// TIA Portal V17 export
// export: Created 2025-03-07T09:23:50.1385037Z, ExportSetting WithDefaults, DisplayName Totally Integrated Automation Portal, DisplayVersion V17 Update 8, DisplayName TIA Portal Openness, DisplayVersion V17 Update 8, DisplayName TIA Portal Version Control Interface, DisplayVersion V17, DisplayName SINAMICS Startdrive Advanced, DisplayVersion V17 SP2, DisplayName SINAMICS Startdrive G110M, G120, G120C, G120D, G120P, G115D, DisplayVersion V17 SP2, DisplayName SINAMICS Startdrive G130, G150, S120, S150, SINAMICS MV, S210, DisplayVersion V17 SP2, DisplayName STEP 7 Professional, DisplayVersion V17 Update 8, DisplayName SINUMERIK ONE STEP 7 Toolbox, DisplayVersion V17 Update 12, DisplayName SINUMERIK 840D sl STEP 7 Toolbox, DisplayVersion V17 Update 12, DisplayName STEP 7 Safety, DisplayVersion V17 Update 6, DisplayName WinCC Advanced, DisplayVersion V17 Update 8
FUNCTION "FC7341_MACHINE_TO_POWDER_INTERLOCK" : Void   // FC7341, LAD
{ S7_Optimized_Access := 'TRUE' }
VERSION : 0.1
// stored: AutoNumber false, IsIECCheckEnabled false, SetENOAutomatically false, UDAEnableTagReadback false
   VAR_TEMP
      "COUNT_FOR _ERROR" : Int;
      EKS_IDENT : Array[0..7] of Char;   // EKS OPERATOR ID
   END_VAR
   VAR CONSTANT
      FC_NUMBER : DInt := 7341;
   END_VAR
BEGIN

REGION Network 1: //////////_GENERAL_//////////
END_REGION

REGION Network 2: LIFE BIT
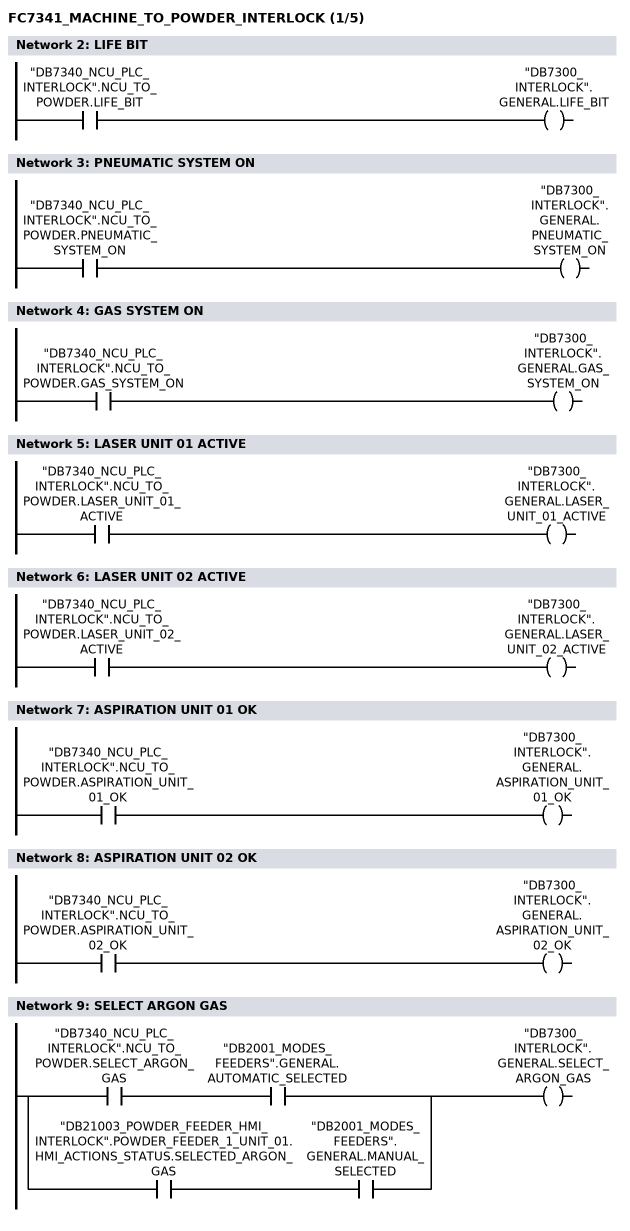
   RUNG wire#powerrail
      Contact( "DB7340_NCU_PLC_INTERLOCK".NCU_TO_POWDER.LIFE_BIT )
      Coil( "DB7300_INTERLOCK".GENERAL.LIFE_BIT )
   END_RUNG
   // the same network as SCL:
   "DB7300_INTERLOCK".GENERAL.LIFE_BIT := "DB7340_NCU_PLC_INTERLOCK".NCU_TO_POWDER.LIFE_BIT;
END_REGION

REGION Network 3: PNEUMATIC SYSTEM ON
   RUNG wire#powerrail
      Contact( "DB7340_NCU_PLC_INTERLOCK".NCU_TO_POWDER.PNEUMATIC_SYSTEM_ON )
      Coil( "DB7300_INTERLOCK".GENERAL.PNEUMATIC_SYSTEM_ON )
   END_RUNG
   // the same network as SCL:
   "DB7300_INTERLOCK".GENERAL.PNEUMATIC_SYSTEM_ON := "DB7340_NCU_PLC_INTERLOCK".NCU_TO_POWDER.PNEUMATIC_SYSTEM_ON;
END_REGION

REGION Network 4: GAS SYSTEM ON
   RUNG wire#powerrail
      Contact( "DB7340_NCU_PLC_INTERLOCK".NCU_TO_POWDER.GAS_SYSTEM_ON )
      Coil( "DB7300_INTERLOCK".GENERAL.GAS_SYSTEM_ON )
   END_RUNG
   // the same network as SCL:
   "DB7300_INTERLOCK".GENERAL.GAS_SYSTEM_ON := "DB7340_NCU_PLC_INTERLOCK".NCU_TO_POWDER.GAS_SYSTEM_ON;
END_REGION

REGION Network 5: LASER UNIT 01 ACTIVE
   RUNG wire#powerrail
      Contact( "DB7340_NCU_PLC_INTERLOCK".NCU_TO_POWDER.LASER_UNIT_01_ACTIVE )
      Coil( "DB7300_INTERLOCK".GENERAL.LASER_UNIT_01_ACTIVE )
   END_RUNG
   // the same network as SCL:
   "DB7300_INTERLOCK".GENERAL.LASER_UNIT_01_ACTIVE := "DB7340_NCU_PLC_INTERLOCK".NCU_TO_POWDER.LASER_UNIT_01_ACTIVE;
END_REGION

REGION Network 6: LASER UNIT 02 ACTIVE
   RUNG wire#powerrail
      Contact( "DB7340_NCU_PLC_INTERLOCK".NCU_TO_POWDER.LASER_UNIT_02_ACTIVE )
      Coil( "DB7300_INTERLOCK".GENERAL.LASER_UNIT_02_ACTIVE )
   END_RUNG
   // the same network as SCL:
   "DB7300_INTERLOCK".GENERAL.LASER_UNIT_02_ACTIVE := "DB7340_NCU_PLC_INTERLOCK".NCU_TO_POWDER.LASER_UNIT_02_ACTIVE;
END_REGION

REGION Network 7: ASPIRATION UNIT 01 OK
   RUNG wire#powerrail
      Contact( "DB7340_NCU_PLC_INTERLOCK".NCU_TO_POWDER.ASPIRATION_UNIT_01_OK )
      Coil( "DB7300_INTERLOCK".GENERAL.ASPIRATION_UNIT_01_OK )
   END_RUNG
   // the same network as SCL:
   "DB7300_INTERLOCK".GENERAL.ASPIRATION_UNIT_01_OK := "DB7340_NCU_PLC_INTERLOCK".NCU_TO_POWDER.ASPIRATION_UNIT_01_OK;
END_REGION

REGION Network 8: ASPIRATION UNIT 02 OK
   RUNG wire#powerrail
      Contact( "DB7340_NCU_PLC_INTERLOCK".NCU_TO_POWDER.ASPIRATION_UNIT_02_OK )
      Coil( "DB7300_INTERLOCK".GENERAL.ASPIRATION_UNIT_02_OK )
   END_RUNG
   // the same network as SCL:
   "DB7300_INTERLOCK".GENERAL.ASPIRATION_UNIT_02_OK := "DB7340_NCU_PLC_INTERLOCK".NCU_TO_POWDER.ASPIRATION_UNIT_02_OK;
END_REGION

REGION Network 9: SELECT ARGON GAS
   RUNG wire#powerrail
      Contact( "DB7340_NCU_PLC_INTERLOCK".NCU_TO_POWDER.SELECT_ARGON_GAS )
      Contact( "DB2001_MODES_FEEDERS".GENERAL.AUTOMATIC_SELECTED )
      wire#w1
      Coil( "DB7300_INTERLOCK".GENERAL.SELECT_ARGON_GAS )
   END_RUNG
   RUNG wire#powerrail
      Contact( "DB21003_POWDER_FEEDER_HMI_INTERLOCK".POWDER_FEEDER_1_UNIT_01.HMI_ACTIONS_STATUS.SELECTED_ARGON_GAS )
      Contact( "DB2001_MODES_FEEDERS".GENERAL.MANUAL_SELECTED )
   END_RUNG wire#w1
   // the same network as SCL:
   "DB7300_INTERLOCK".GENERAL.SELECT_ARGON_GAS := ("DB7340_NCU_PLC_INTERLOCK".NCU_TO_POWDER.SELECT_ARGON_GAS AND "DB2001_MODES_FEEDERS".GENERAL.AUTOMATIC_SELECTED) OR ("DB21003_POWDER_FEEDER_HMI_INTERLOCK".POWDER_FEEDER_1_UNIT_01.HMI_ACTIONS_STATUS.SELECTED_ARGON_GAS AND "DB2001_MODES_FEEDERS".GENERAL.MANUAL_SELECTED);
END_REGION

REGION Network 10: SELECT NITROGEN GAS
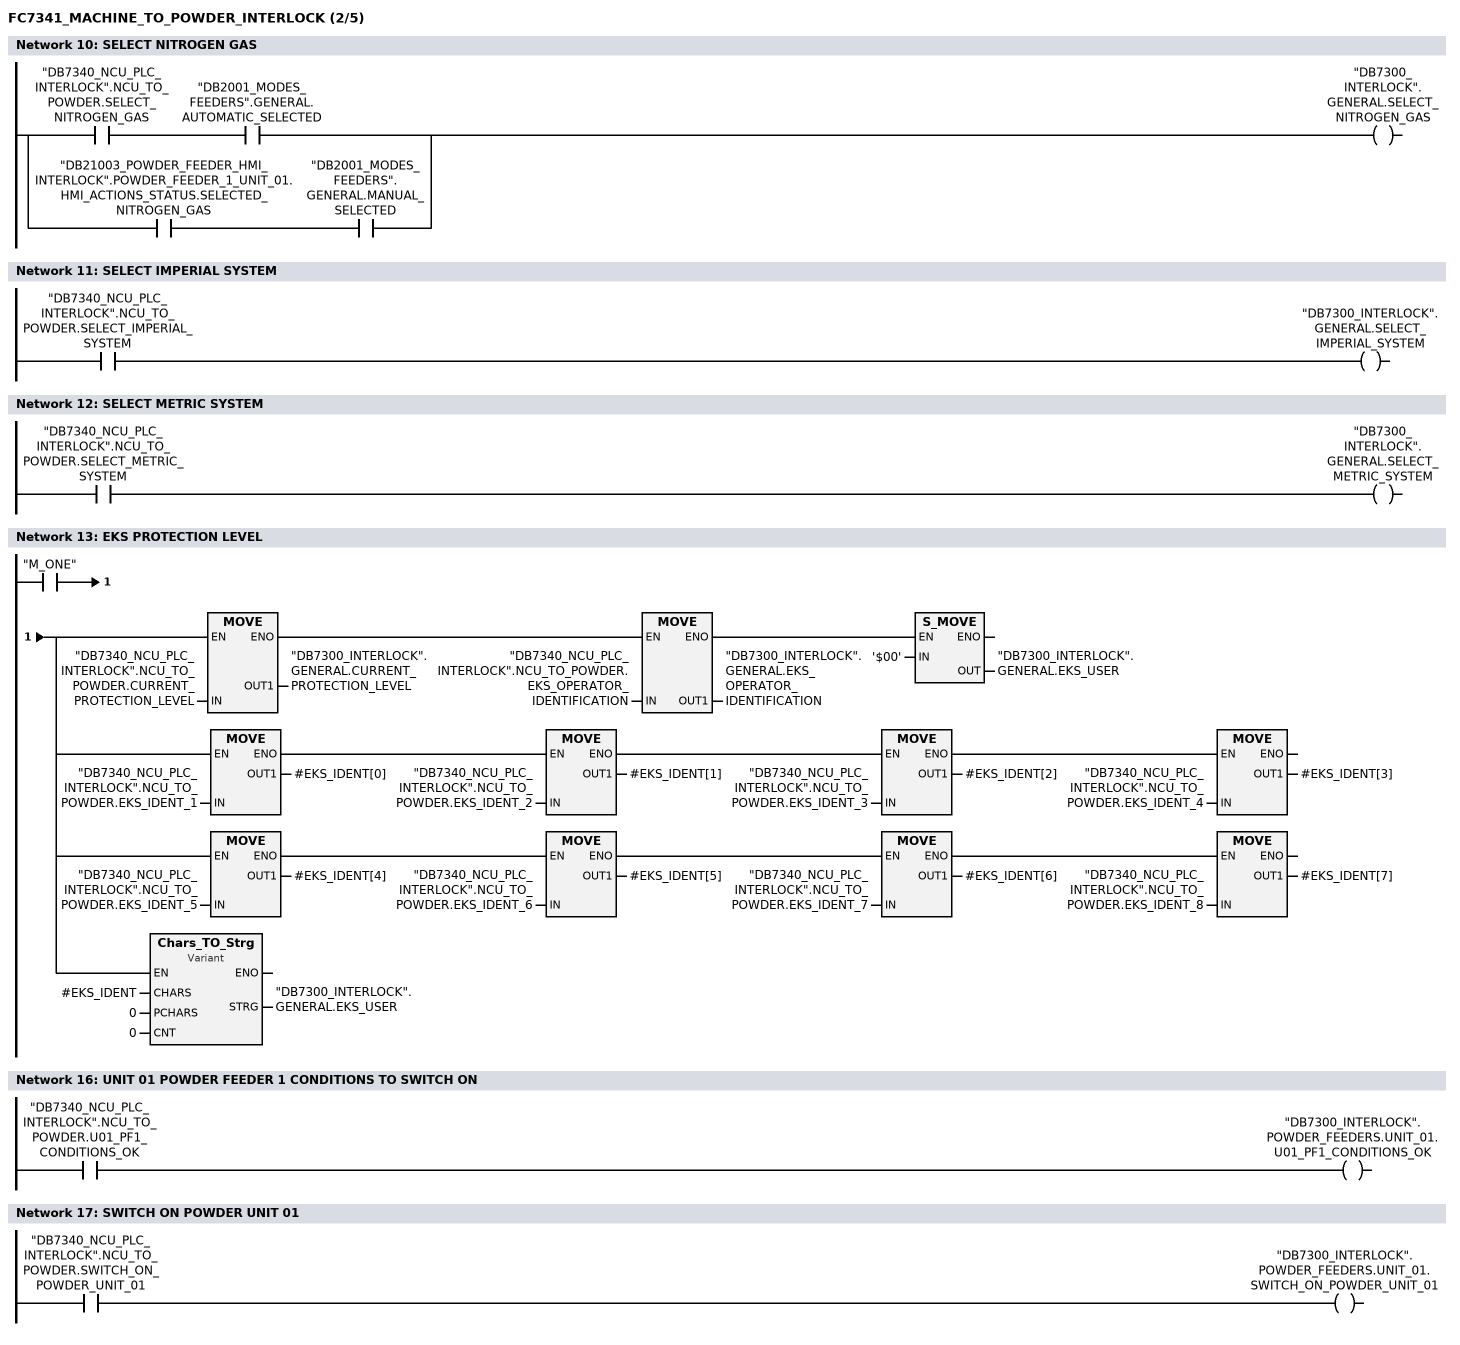
   RUNG wire#powerrail
      Contact( "DB7340_NCU_PLC_INTERLOCK".NCU_TO_POWDER.SELECT_NITROGEN_GAS )
      Contact( "DB2001_MODES_FEEDERS".GENERAL.AUTOMATIC_SELECTED )
      wire#w1
      Coil( "DB7300_INTERLOCK".GENERAL.SELECT_NITROGEN_GAS )
   END_RUNG
   RUNG wire#powerrail
      Contact( "DB21003_POWDER_FEEDER_HMI_INTERLOCK".POWDER_FEEDER_1_UNIT_01.HMI_ACTIONS_STATUS.SELECTED_NITROGEN_GAS )
      Contact( "DB2001_MODES_FEEDERS".GENERAL.MANUAL_SELECTED )
   END_RUNG wire#w1
   // the same network as SCL:
   "DB7300_INTERLOCK".GENERAL.SELECT_NITROGEN_GAS := ("DB7340_NCU_PLC_INTERLOCK".NCU_TO_POWDER.SELECT_NITROGEN_GAS AND "DB2001_MODES_FEEDERS".GENERAL.AUTOMATIC_SELECTED) OR ("DB21003_POWDER_FEEDER_HMI_INTERLOCK".POWDER_FEEDER_1_UNIT_01.HMI_ACTIONS_STATUS.SELECTED_NITROGEN_GAS AND "DB2001_MODES_FEEDERS".GENERAL.MANUAL_SELECTED);
END_REGION

REGION Network 11: SELECT IMPERIAL SYSTEM
   RUNG wire#powerrail
      Contact( "DB7340_NCU_PLC_INTERLOCK".NCU_TO_POWDER.SELECT_IMPERIAL_SYSTEM )
      Coil( "DB7300_INTERLOCK".GENERAL.SELECT_IMPERIAL_SYSTEM )
   END_RUNG
   // the same network as SCL:
   "DB7300_INTERLOCK".GENERAL.SELECT_IMPERIAL_SYSTEM := "DB7340_NCU_PLC_INTERLOCK".NCU_TO_POWDER.SELECT_IMPERIAL_SYSTEM;
END_REGION

REGION Network 12: SELECT METRIC SYSTEM
   RUNG wire#powerrail
      Contact( "DB7340_NCU_PLC_INTERLOCK".NCU_TO_POWDER.SELECT_METRIC_SYSTEM )
      Coil( "DB7300_INTERLOCK".GENERAL.SELECT_METRIC_SYSTEM )
   END_RUNG
   // the same network as SCL:
   "DB7300_INTERLOCK".GENERAL.SELECT_METRIC_SYSTEM := "DB7340_NCU_PLC_INTERLOCK".NCU_TO_POWDER.SELECT_METRIC_SYSTEM;
END_REGION

REGION Network 13: EKS PROTECTION LEVEL
   RUNG wire#powerrail
      Contact( "M_ONE" )
      wire#w1
      Move(in := "DB7340_NCU_PLC_INTERLOCK".NCU_TO_POWDER.CURRENT_PROTECTION_LEVEL, out1 => "DB7300_INTERLOCK".GENERAL.CURRENT_PROTECTION_LEVEL)
      Move(in := "DB7340_NCU_PLC_INTERLOCK".NCU_TO_POWDER.EKS_OPERATOR_IDENTIFICATION, out1 => "DB7300_INTERLOCK".GENERAL.EKS_OPERATOR_IDENTIFICATION)
      S_Move(in := '$00', out => "DB7300_INTERLOCK".GENERAL.EKS_USER)
   END_RUNG
   RUNG wire#w1
      Move(in := "DB7340_NCU_PLC_INTERLOCK".NCU_TO_POWDER.EKS_IDENT_1, out1 => #EKS_IDENT[0])
      Move(in := "DB7340_NCU_PLC_INTERLOCK".NCU_TO_POWDER.EKS_IDENT_2, out1 => #EKS_IDENT[1])
      Move(in := "DB7340_NCU_PLC_INTERLOCK".NCU_TO_POWDER.EKS_IDENT_3, out1 => #EKS_IDENT[2])
      Move(in := "DB7340_NCU_PLC_INTERLOCK".NCU_TO_POWDER.EKS_IDENT_4, out1 => #EKS_IDENT[3])
   END_RUNG
   RUNG wire#w1
      Move(in := "DB7340_NCU_PLC_INTERLOCK".NCU_TO_POWDER.EKS_IDENT_5, out1 => #EKS_IDENT[4])
      Move(in := "DB7340_NCU_PLC_INTERLOCK".NCU_TO_POWDER.EKS_IDENT_6, out1 => #EKS_IDENT[5])
      Move(in := "DB7340_NCU_PLC_INTERLOCK".NCU_TO_POWDER.EKS_IDENT_7, out1 => #EKS_IDENT[6])
      Move(in := "DB7340_NCU_PLC_INTERLOCK".NCU_TO_POWDER.EKS_IDENT_8, out1 => #EKS_IDENT[7])
   END_RUNG
   RUNG wire#w1
      { S7_Templates := "[ptr_type := Variant, str_type := String]" } Chars_TO_Strg(Chars := #EKS_IDENT, pChars := 0, Cnt := 0, Strg => "DB7300_INTERLOCK".GENERAL.EKS_USER)
   END_RUNG
   // the same network as SCL:
   IF "M_ONE" THEN
       "DB7300_INTERLOCK".GENERAL.CURRENT_PROTECTION_LEVEL := "DB7340_NCU_PLC_INTERLOCK".NCU_TO_POWDER.CURRENT_PROTECTION_LEVEL;
       "DB7300_INTERLOCK".GENERAL.EKS_OPERATOR_IDENTIFICATION := "DB7340_NCU_PLC_INTERLOCK".NCU_TO_POWDER.EKS_OPERATOR_IDENTIFICATION;
       "DB7300_INTERLOCK".GENERAL.EKS_USER := '$00';
       #EKS_IDENT[0] := "DB7340_NCU_PLC_INTERLOCK".NCU_TO_POWDER.EKS_IDENT_1;
       #EKS_IDENT[1] := "DB7340_NCU_PLC_INTERLOCK".NCU_TO_POWDER.EKS_IDENT_2;
       #EKS_IDENT[2] := "DB7340_NCU_PLC_INTERLOCK".NCU_TO_POWDER.EKS_IDENT_3;
       #EKS_IDENT[3] := "DB7340_NCU_PLC_INTERLOCK".NCU_TO_POWDER.EKS_IDENT_4;
       #EKS_IDENT[4] := "DB7340_NCU_PLC_INTERLOCK".NCU_TO_POWDER.EKS_IDENT_5;
       #EKS_IDENT[5] := "DB7340_NCU_PLC_INTERLOCK".NCU_TO_POWDER.EKS_IDENT_6;
       #EKS_IDENT[6] := "DB7340_NCU_PLC_INTERLOCK".NCU_TO_POWDER.EKS_IDENT_7;
       #EKS_IDENT[7] := "DB7340_NCU_PLC_INTERLOCK".NCU_TO_POWDER.EKS_IDENT_8;
       Chars_TO_Strg(Chars := #EKS_IDENT, pChars := 0, Cnt := 0, Strg => "DB7300_INTERLOCK".GENERAL.EKS_USER);
   END_IF;
END_REGION

REGION Network 14: //////////_POWDER_FEEDERS_//////////
END_REGION

REGION Network 15: /////_UNIT_01_/////
END_REGION

REGION Network 16: UNIT 01 POWDER FEEDER 1 CONDITIONS TO SWITCH ON
   RUNG wire#powerrail
      Contact( "DB7340_NCU_PLC_INTERLOCK".NCU_TO_POWDER.U01_PF1_CONDITIONS_OK )
      Coil( "DB7300_INTERLOCK".POWDER_FEEDERS.UNIT_01.U01_PF1_CONDITIONS_OK )
   END_RUNG
   // the same network as SCL:
   "DB7300_INTERLOCK".POWDER_FEEDERS.UNIT_01.U01_PF1_CONDITIONS_OK := "DB7340_NCU_PLC_INTERLOCK".NCU_TO_POWDER.U01_PF1_CONDITIONS_OK;
END_REGION

REGION Network 17: SWITCH ON POWDER UNIT 01
   RUNG wire#powerrail
      Contact( "DB7340_NCU_PLC_INTERLOCK".NCU_TO_POWDER.SWITCH_ON_POWDER_UNIT_01 )
      Coil( "DB7300_INTERLOCK".POWDER_FEEDERS.UNIT_01.SWITCH_ON_POWDER_UNIT_01 )
   END_RUNG
   // the same network as SCL:
   "DB7300_INTERLOCK".POWDER_FEEDERS.UNIT_01.SWITCH_ON_POWDER_UNIT_01 := "DB7340_NCU_PLC_INTERLOCK".NCU_TO_POWDER.SWITCH_ON_POWDER_UNIT_01;
END_REGION

REGION Network 18: SWITCH OFF POWDER UNIT 01
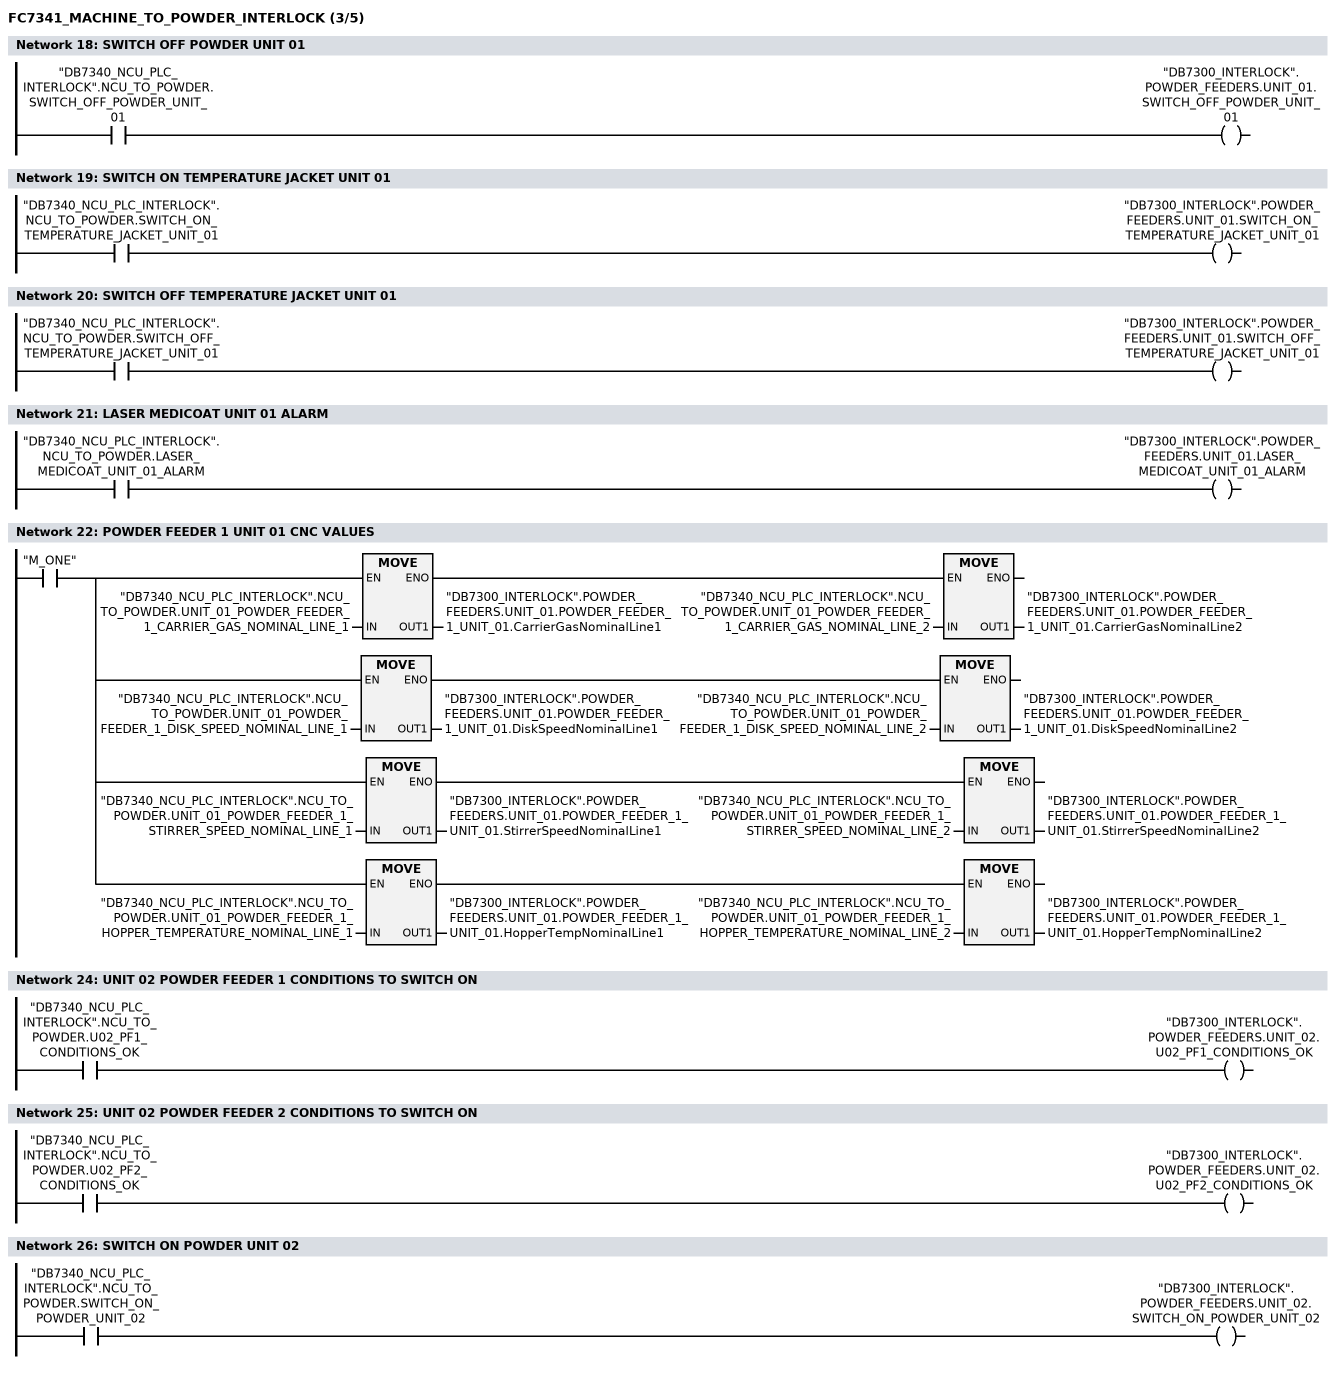
   RUNG wire#powerrail
      Contact( "DB7340_NCU_PLC_INTERLOCK".NCU_TO_POWDER.SWITCH_OFF_POWDER_UNIT_01 )
      Coil( "DB7300_INTERLOCK".POWDER_FEEDERS.UNIT_01.SWITCH_OFF_POWDER_UNIT_01 )
   END_RUNG
   // the same network as SCL:
   "DB7300_INTERLOCK".POWDER_FEEDERS.UNIT_01.SWITCH_OFF_POWDER_UNIT_01 := "DB7340_NCU_PLC_INTERLOCK".NCU_TO_POWDER.SWITCH_OFF_POWDER_UNIT_01;
END_REGION

REGION Network 19: SWITCH ON TEMPERATURE JACKET UNIT 01
   RUNG wire#powerrail
      Contact( "DB7340_NCU_PLC_INTERLOCK".NCU_TO_POWDER.SWITCH_ON_TEMPERATURE_JACKET_UNIT_01 )
      Coil( "DB7300_INTERLOCK".POWDER_FEEDERS.UNIT_01.SWITCH_ON_TEMPERATURE_JACKET_UNIT_01 )
   END_RUNG
   // the same network as SCL:
   "DB7300_INTERLOCK".POWDER_FEEDERS.UNIT_01.SWITCH_ON_TEMPERATURE_JACKET_UNIT_01 := "DB7340_NCU_PLC_INTERLOCK".NCU_TO_POWDER.SWITCH_ON_TEMPERATURE_JACKET_UNIT_01;
END_REGION

REGION Network 20: SWITCH OFF TEMPERATURE JACKET UNIT 01
   RUNG wire#powerrail
      Contact( "DB7340_NCU_PLC_INTERLOCK".NCU_TO_POWDER.SWITCH_OFF_TEMPERATURE_JACKET_UNIT_01 )
      Coil( "DB7300_INTERLOCK".POWDER_FEEDERS.UNIT_01.SWITCH_OFF_TEMPERATURE_JACKET_UNIT_01 )
   END_RUNG
   // the same network as SCL:
   "DB7300_INTERLOCK".POWDER_FEEDERS.UNIT_01.SWITCH_OFF_TEMPERATURE_JACKET_UNIT_01 := "DB7340_NCU_PLC_INTERLOCK".NCU_TO_POWDER.SWITCH_OFF_TEMPERATURE_JACKET_UNIT_01;
END_REGION

REGION Network 21: LASER MEDICOAT UNIT 01 ALARM
   RUNG wire#powerrail
      Contact( "DB7340_NCU_PLC_INTERLOCK".NCU_TO_POWDER.LASER_MEDICOAT_UNIT_01_ALARM )
      Coil( "DB7300_INTERLOCK".POWDER_FEEDERS.UNIT_01.LASER_MEDICOAT_UNIT_01_ALARM )
   END_RUNG
   // the same network as SCL:
   "DB7300_INTERLOCK".POWDER_FEEDERS.UNIT_01.LASER_MEDICOAT_UNIT_01_ALARM := "DB7340_NCU_PLC_INTERLOCK".NCU_TO_POWDER.LASER_MEDICOAT_UNIT_01_ALARM;
END_REGION

REGION Network 22: POWDER FEEDER 1 UNIT 01 CNC VALUES
   RUNG wire#powerrail
      Contact( "M_ONE" )
      wire#w1
      Move(in := "DB7340_NCU_PLC_INTERLOCK".NCU_TO_POWDER.UNIT_01_POWDER_FEEDER_1_CARRIER_GAS_NOMINAL_LINE_1, out1 => "DB7300_INTERLOCK".POWDER_FEEDERS.UNIT_01.POWDER_FEEDER_1_UNIT_01.CarrierGasNominalLine1)
      Move(in := "DB7340_NCU_PLC_INTERLOCK".NCU_TO_POWDER.UNIT_01_POWDER_FEEDER_1_CARRIER_GAS_NOMINAL_LINE_2, out1 => "DB7300_INTERLOCK".POWDER_FEEDERS.UNIT_01.POWDER_FEEDER_1_UNIT_01.CarrierGasNominalLine2)
   END_RUNG
   RUNG wire#w1
      Move(in := "DB7340_NCU_PLC_INTERLOCK".NCU_TO_POWDER.UNIT_01_POWDER_FEEDER_1_DISK_SPEED_NOMINAL_LINE_1, out1 => "DB7300_INTERLOCK".POWDER_FEEDERS.UNIT_01.POWDER_FEEDER_1_UNIT_01.DiskSpeedNominalLine1)
      Move(in := "DB7340_NCU_PLC_INTERLOCK".NCU_TO_POWDER.UNIT_01_POWDER_FEEDER_1_DISK_SPEED_NOMINAL_LINE_2, out1 => "DB7300_INTERLOCK".POWDER_FEEDERS.UNIT_01.POWDER_FEEDER_1_UNIT_01.DiskSpeedNominalLine2)
   END_RUNG
   RUNG wire#w1
      Move(in := "DB7340_NCU_PLC_INTERLOCK".NCU_TO_POWDER.UNIT_01_POWDER_FEEDER_1_STIRRER_SPEED_NOMINAL_LINE_1, out1 => "DB7300_INTERLOCK".POWDER_FEEDERS.UNIT_01.POWDER_FEEDER_1_UNIT_01.StirrerSpeedNominalLine1)
      Move(in := "DB7340_NCU_PLC_INTERLOCK".NCU_TO_POWDER.UNIT_01_POWDER_FEEDER_1_STIRRER_SPEED_NOMINAL_LINE_2, out1 => "DB7300_INTERLOCK".POWDER_FEEDERS.UNIT_01.POWDER_FEEDER_1_UNIT_01.StirrerSpeedNominalLine2)
   END_RUNG
   RUNG wire#w1
      Move(in := "DB7340_NCU_PLC_INTERLOCK".NCU_TO_POWDER.UNIT_01_POWDER_FEEDER_1_HOPPER_TEMPERATURE_NOMINAL_LINE_1, out1 => "DB7300_INTERLOCK".POWDER_FEEDERS.UNIT_01.POWDER_FEEDER_1_UNIT_01.HopperTempNominalLine1)
      Move(in := "DB7340_NCU_PLC_INTERLOCK".NCU_TO_POWDER.UNIT_01_POWDER_FEEDER_1_HOPPER_TEMPERATURE_NOMINAL_LINE_2, out1 => "DB7300_INTERLOCK".POWDER_FEEDERS.UNIT_01.POWDER_FEEDER_1_UNIT_01.HopperTempNominalLine2)
   END_RUNG
   // the same network as SCL:
   IF "M_ONE" THEN
       "DB7300_INTERLOCK".POWDER_FEEDERS.UNIT_01.POWDER_FEEDER_1_UNIT_01.CarrierGasNominalLine1 := "DB7340_NCU_PLC_INTERLOCK".NCU_TO_POWDER.UNIT_01_POWDER_FEEDER_1_CARRIER_GAS_NOMINAL_LINE_1;
       "DB7300_INTERLOCK".POWDER_FEEDERS.UNIT_01.POWDER_FEEDER_1_UNIT_01.CarrierGasNominalLine2 := "DB7340_NCU_PLC_INTERLOCK".NCU_TO_POWDER.UNIT_01_POWDER_FEEDER_1_CARRIER_GAS_NOMINAL_LINE_2;
       "DB7300_INTERLOCK".POWDER_FEEDERS.UNIT_01.POWDER_FEEDER_1_UNIT_01.DiskSpeedNominalLine1 := "DB7340_NCU_PLC_INTERLOCK".NCU_TO_POWDER.UNIT_01_POWDER_FEEDER_1_DISK_SPEED_NOMINAL_LINE_1;
       "DB7300_INTERLOCK".POWDER_FEEDERS.UNIT_01.POWDER_FEEDER_1_UNIT_01.DiskSpeedNominalLine2 := "DB7340_NCU_PLC_INTERLOCK".NCU_TO_POWDER.UNIT_01_POWDER_FEEDER_1_DISK_SPEED_NOMINAL_LINE_2;
       "DB7300_INTERLOCK".POWDER_FEEDERS.UNIT_01.POWDER_FEEDER_1_UNIT_01.StirrerSpeedNominalLine1 := "DB7340_NCU_PLC_INTERLOCK".NCU_TO_POWDER.UNIT_01_POWDER_FEEDER_1_STIRRER_SPEED_NOMINAL_LINE_1;
       "DB7300_INTERLOCK".POWDER_FEEDERS.UNIT_01.POWDER_FEEDER_1_UNIT_01.StirrerSpeedNominalLine2 := "DB7340_NCU_PLC_INTERLOCK".NCU_TO_POWDER.UNIT_01_POWDER_FEEDER_1_STIRRER_SPEED_NOMINAL_LINE_2;
       "DB7300_INTERLOCK".POWDER_FEEDERS.UNIT_01.POWDER_FEEDER_1_UNIT_01.HopperTempNominalLine1 := "DB7340_NCU_PLC_INTERLOCK".NCU_TO_POWDER.UNIT_01_POWDER_FEEDER_1_HOPPER_TEMPERATURE_NOMINAL_LINE_1;
       "DB7300_INTERLOCK".POWDER_FEEDERS.UNIT_01.POWDER_FEEDER_1_UNIT_01.HopperTempNominalLine2 := "DB7340_NCU_PLC_INTERLOCK".NCU_TO_POWDER.UNIT_01_POWDER_FEEDER_1_HOPPER_TEMPERATURE_NOMINAL_LINE_2;
   END_IF;
END_REGION

REGION Network 23: /////_UNIT_02_/////
END_REGION

REGION Network 24: UNIT 02 POWDER FEEDER 1 CONDITIONS TO SWITCH ON
   RUNG wire#powerrail
      Contact( "DB7340_NCU_PLC_INTERLOCK".NCU_TO_POWDER.U02_PF1_CONDITIONS_OK )
      Coil( "DB7300_INTERLOCK".POWDER_FEEDERS.UNIT_02.U02_PF1_CONDITIONS_OK )
   END_RUNG
   // the same network as SCL:
   "DB7300_INTERLOCK".POWDER_FEEDERS.UNIT_02.U02_PF1_CONDITIONS_OK := "DB7340_NCU_PLC_INTERLOCK".NCU_TO_POWDER.U02_PF1_CONDITIONS_OK;
END_REGION

REGION Network 25: UNIT 02 POWDER FEEDER 2 CONDITIONS TO SWITCH ON
   RUNG wire#powerrail
      Contact( "DB7340_NCU_PLC_INTERLOCK".NCU_TO_POWDER.U02_PF2_CONDITIONS_OK )
      Coil( "DB7300_INTERLOCK".POWDER_FEEDERS.UNIT_02.U02_PF2_CONDITIONS_OK )
   END_RUNG
   // the same network as SCL:
   "DB7300_INTERLOCK".POWDER_FEEDERS.UNIT_02.U02_PF2_CONDITIONS_OK := "DB7340_NCU_PLC_INTERLOCK".NCU_TO_POWDER.U02_PF2_CONDITIONS_OK;
END_REGION

REGION Network 26: SWITCH ON POWDER UNIT 02
   RUNG wire#powerrail
      Contact( "DB7340_NCU_PLC_INTERLOCK".NCU_TO_POWDER.SWITCH_ON_POWDER_UNIT_02 )
      Coil( "DB7300_INTERLOCK".POWDER_FEEDERS.UNIT_02.SWITCH_ON_POWDER_UNIT_02 )
   END_RUNG
   // the same network as SCL:
   "DB7300_INTERLOCK".POWDER_FEEDERS.UNIT_02.SWITCH_ON_POWDER_UNIT_02 := "DB7340_NCU_PLC_INTERLOCK".NCU_TO_POWDER.SWITCH_ON_POWDER_UNIT_02;
END_REGION

REGION Network 27: SWITCH OFF POWDER UNIT 02
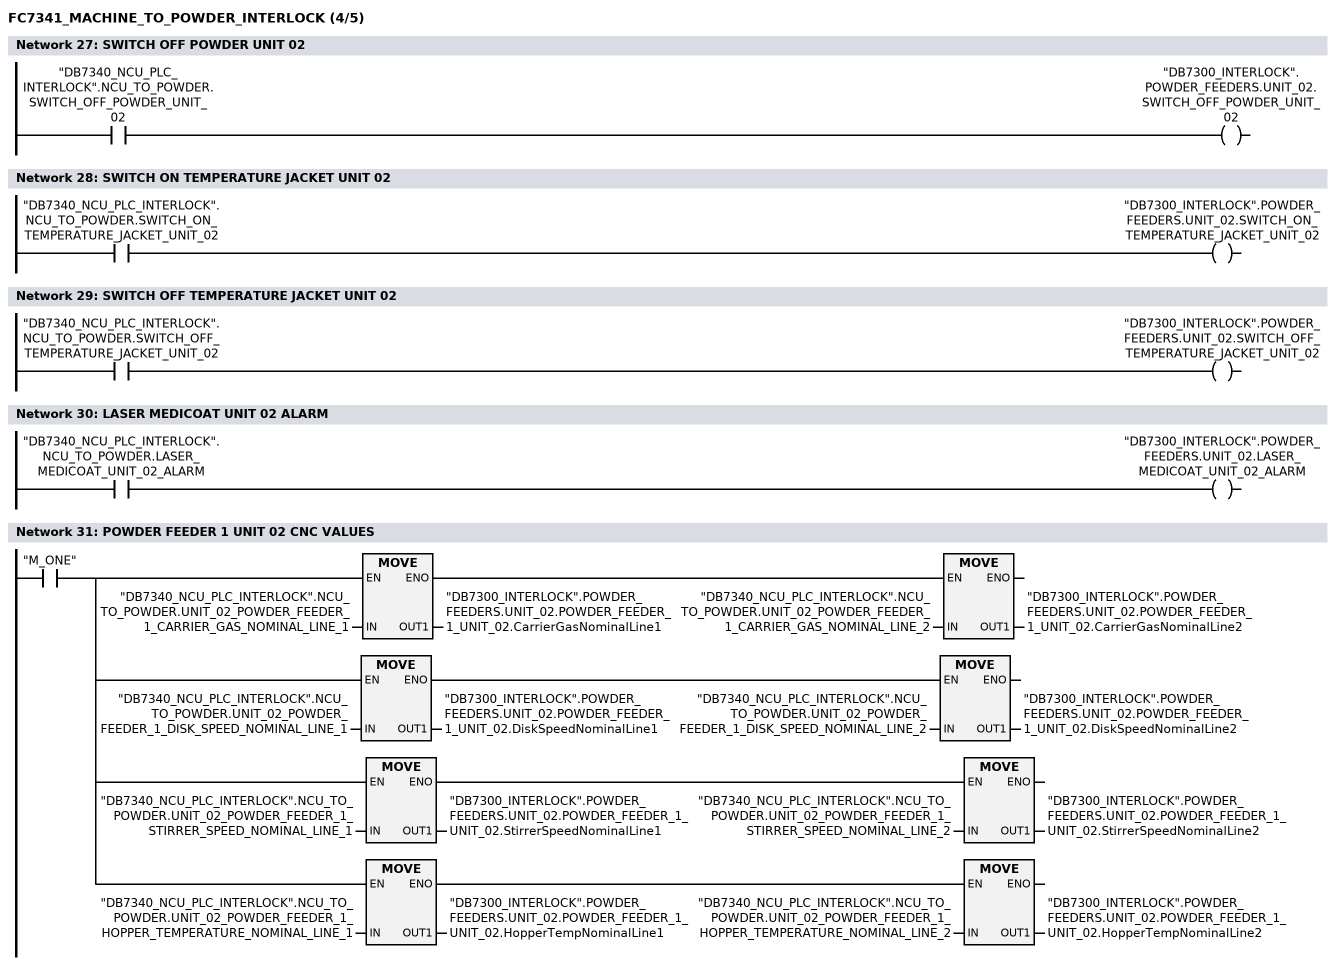
   RUNG wire#powerrail
      Contact( "DB7340_NCU_PLC_INTERLOCK".NCU_TO_POWDER.SWITCH_OFF_POWDER_UNIT_02 )
      Coil( "DB7300_INTERLOCK".POWDER_FEEDERS.UNIT_02.SWITCH_OFF_POWDER_UNIT_02 )
   END_RUNG
   // the same network as SCL:
   "DB7300_INTERLOCK".POWDER_FEEDERS.UNIT_02.SWITCH_OFF_POWDER_UNIT_02 := "DB7340_NCU_PLC_INTERLOCK".NCU_TO_POWDER.SWITCH_OFF_POWDER_UNIT_02;
END_REGION

REGION Network 28: SWITCH ON TEMPERATURE JACKET UNIT 02
   RUNG wire#powerrail
      Contact( "DB7340_NCU_PLC_INTERLOCK".NCU_TO_POWDER.SWITCH_ON_TEMPERATURE_JACKET_UNIT_02 )
      Coil( "DB7300_INTERLOCK".POWDER_FEEDERS.UNIT_02.SWITCH_ON_TEMPERATURE_JACKET_UNIT_02 )
   END_RUNG
   // the same network as SCL:
   "DB7300_INTERLOCK".POWDER_FEEDERS.UNIT_02.SWITCH_ON_TEMPERATURE_JACKET_UNIT_02 := "DB7340_NCU_PLC_INTERLOCK".NCU_TO_POWDER.SWITCH_ON_TEMPERATURE_JACKET_UNIT_02;
END_REGION

REGION Network 29: SWITCH OFF TEMPERATURE JACKET UNIT 02
   RUNG wire#powerrail
      Contact( "DB7340_NCU_PLC_INTERLOCK".NCU_TO_POWDER.SWITCH_OFF_TEMPERATURE_JACKET_UNIT_02 )
      Coil( "DB7300_INTERLOCK".POWDER_FEEDERS.UNIT_02.SWITCH_OFF_TEMPERATURE_JACKET_UNIT_02 )
   END_RUNG
   // the same network as SCL:
   "DB7300_INTERLOCK".POWDER_FEEDERS.UNIT_02.SWITCH_OFF_TEMPERATURE_JACKET_UNIT_02 := "DB7340_NCU_PLC_INTERLOCK".NCU_TO_POWDER.SWITCH_OFF_TEMPERATURE_JACKET_UNIT_02;
END_REGION

REGION Network 30: LASER MEDICOAT UNIT 02 ALARM
   RUNG wire#powerrail
      Contact( "DB7340_NCU_PLC_INTERLOCK".NCU_TO_POWDER.LASER_MEDICOAT_UNIT_02_ALARM )
      Coil( "DB7300_INTERLOCK".POWDER_FEEDERS.UNIT_02.LASER_MEDICOAT_UNIT_02_ALARM )
   END_RUNG
   // the same network as SCL:
   "DB7300_INTERLOCK".POWDER_FEEDERS.UNIT_02.LASER_MEDICOAT_UNIT_02_ALARM := "DB7340_NCU_PLC_INTERLOCK".NCU_TO_POWDER.LASER_MEDICOAT_UNIT_02_ALARM;
END_REGION

REGION Network 31: POWDER FEEDER 1 UNIT 02 CNC VALUES
   RUNG wire#powerrail
      Contact( "M_ONE" )
      wire#w1
      Move(in := "DB7340_NCU_PLC_INTERLOCK".NCU_TO_POWDER.UNIT_02_POWDER_FEEDER_1_CARRIER_GAS_NOMINAL_LINE_1, out1 => "DB7300_INTERLOCK".POWDER_FEEDERS.UNIT_02.POWDER_FEEDER_1_UNIT_02.CarrierGasNominalLine1)
      Move(in := "DB7340_NCU_PLC_INTERLOCK".NCU_TO_POWDER.UNIT_02_POWDER_FEEDER_1_CARRIER_GAS_NOMINAL_LINE_2, out1 => "DB7300_INTERLOCK".POWDER_FEEDERS.UNIT_02.POWDER_FEEDER_1_UNIT_02.CarrierGasNominalLine2)
   END_RUNG
   RUNG wire#w1
      Move(in := "DB7340_NCU_PLC_INTERLOCK".NCU_TO_POWDER.UNIT_02_POWDER_FEEDER_1_DISK_SPEED_NOMINAL_LINE_1, out1 => "DB7300_INTERLOCK".POWDER_FEEDERS.UNIT_02.POWDER_FEEDER_1_UNIT_02.DiskSpeedNominalLine1)
      Move(in := "DB7340_NCU_PLC_INTERLOCK".NCU_TO_POWDER.UNIT_02_POWDER_FEEDER_1_DISK_SPEED_NOMINAL_LINE_2, out1 => "DB7300_INTERLOCK".POWDER_FEEDERS.UNIT_02.POWDER_FEEDER_1_UNIT_02.DiskSpeedNominalLine2)
   END_RUNG
   RUNG wire#w1
      Move(in := "DB7340_NCU_PLC_INTERLOCK".NCU_TO_POWDER.UNIT_02_POWDER_FEEDER_1_STIRRER_SPEED_NOMINAL_LINE_1, out1 => "DB7300_INTERLOCK".POWDER_FEEDERS.UNIT_02.POWDER_FEEDER_1_UNIT_02.StirrerSpeedNominalLine1)
      Move(in := "DB7340_NCU_PLC_INTERLOCK".NCU_TO_POWDER.UNIT_02_POWDER_FEEDER_1_STIRRER_SPEED_NOMINAL_LINE_2, out1 => "DB7300_INTERLOCK".POWDER_FEEDERS.UNIT_02.POWDER_FEEDER_1_UNIT_02.StirrerSpeedNominalLine2)
   END_RUNG
   RUNG wire#w1
      Move(in := "DB7340_NCU_PLC_INTERLOCK".NCU_TO_POWDER.UNIT_02_POWDER_FEEDER_1_HOPPER_TEMPERATURE_NOMINAL_LINE_1, out1 => "DB7300_INTERLOCK".POWDER_FEEDERS.UNIT_02.POWDER_FEEDER_1_UNIT_02.HopperTempNominalLine1)
      Move(in := "DB7340_NCU_PLC_INTERLOCK".NCU_TO_POWDER.UNIT_02_POWDER_FEEDER_1_HOPPER_TEMPERATURE_NOMINAL_LINE_2, out1 => "DB7300_INTERLOCK".POWDER_FEEDERS.UNIT_02.POWDER_FEEDER_1_UNIT_02.HopperTempNominalLine2)
   END_RUNG
   // the same network as SCL:
   IF "M_ONE" THEN
       "DB7300_INTERLOCK".POWDER_FEEDERS.UNIT_02.POWDER_FEEDER_1_UNIT_02.CarrierGasNominalLine1 := "DB7340_NCU_PLC_INTERLOCK".NCU_TO_POWDER.UNIT_02_POWDER_FEEDER_1_CARRIER_GAS_NOMINAL_LINE_1;
       "DB7300_INTERLOCK".POWDER_FEEDERS.UNIT_02.POWDER_FEEDER_1_UNIT_02.CarrierGasNominalLine2 := "DB7340_NCU_PLC_INTERLOCK".NCU_TO_POWDER.UNIT_02_POWDER_FEEDER_1_CARRIER_GAS_NOMINAL_LINE_2;
       "DB7300_INTERLOCK".POWDER_FEEDERS.UNIT_02.POWDER_FEEDER_1_UNIT_02.DiskSpeedNominalLine1 := "DB7340_NCU_PLC_INTERLOCK".NCU_TO_POWDER.UNIT_02_POWDER_FEEDER_1_DISK_SPEED_NOMINAL_LINE_1;
       "DB7300_INTERLOCK".POWDER_FEEDERS.UNIT_02.POWDER_FEEDER_1_UNIT_02.DiskSpeedNominalLine2 := "DB7340_NCU_PLC_INTERLOCK".NCU_TO_POWDER.UNIT_02_POWDER_FEEDER_1_DISK_SPEED_NOMINAL_LINE_2;
       "DB7300_INTERLOCK".POWDER_FEEDERS.UNIT_02.POWDER_FEEDER_1_UNIT_02.StirrerSpeedNominalLine1 := "DB7340_NCU_PLC_INTERLOCK".NCU_TO_POWDER.UNIT_02_POWDER_FEEDER_1_STIRRER_SPEED_NOMINAL_LINE_1;
       "DB7300_INTERLOCK".POWDER_FEEDERS.UNIT_02.POWDER_FEEDER_1_UNIT_02.StirrerSpeedNominalLine2 := "DB7340_NCU_PLC_INTERLOCK".NCU_TO_POWDER.UNIT_02_POWDER_FEEDER_1_STIRRER_SPEED_NOMINAL_LINE_2;
       "DB7300_INTERLOCK".POWDER_FEEDERS.UNIT_02.POWDER_FEEDER_1_UNIT_02.HopperTempNominalLine1 := "DB7340_NCU_PLC_INTERLOCK".NCU_TO_POWDER.UNIT_02_POWDER_FEEDER_1_HOPPER_TEMPERATURE_NOMINAL_LINE_1;
       "DB7300_INTERLOCK".POWDER_FEEDERS.UNIT_02.POWDER_FEEDER_1_UNIT_02.HopperTempNominalLine2 := "DB7340_NCU_PLC_INTERLOCK".NCU_TO_POWDER.UNIT_02_POWDER_FEEDER_1_HOPPER_TEMPERATURE_NOMINAL_LINE_2;
   END_IF;
END_REGION

REGION Network 32: POWDER FEEDER 2 UNIT 02 CNC VALUES
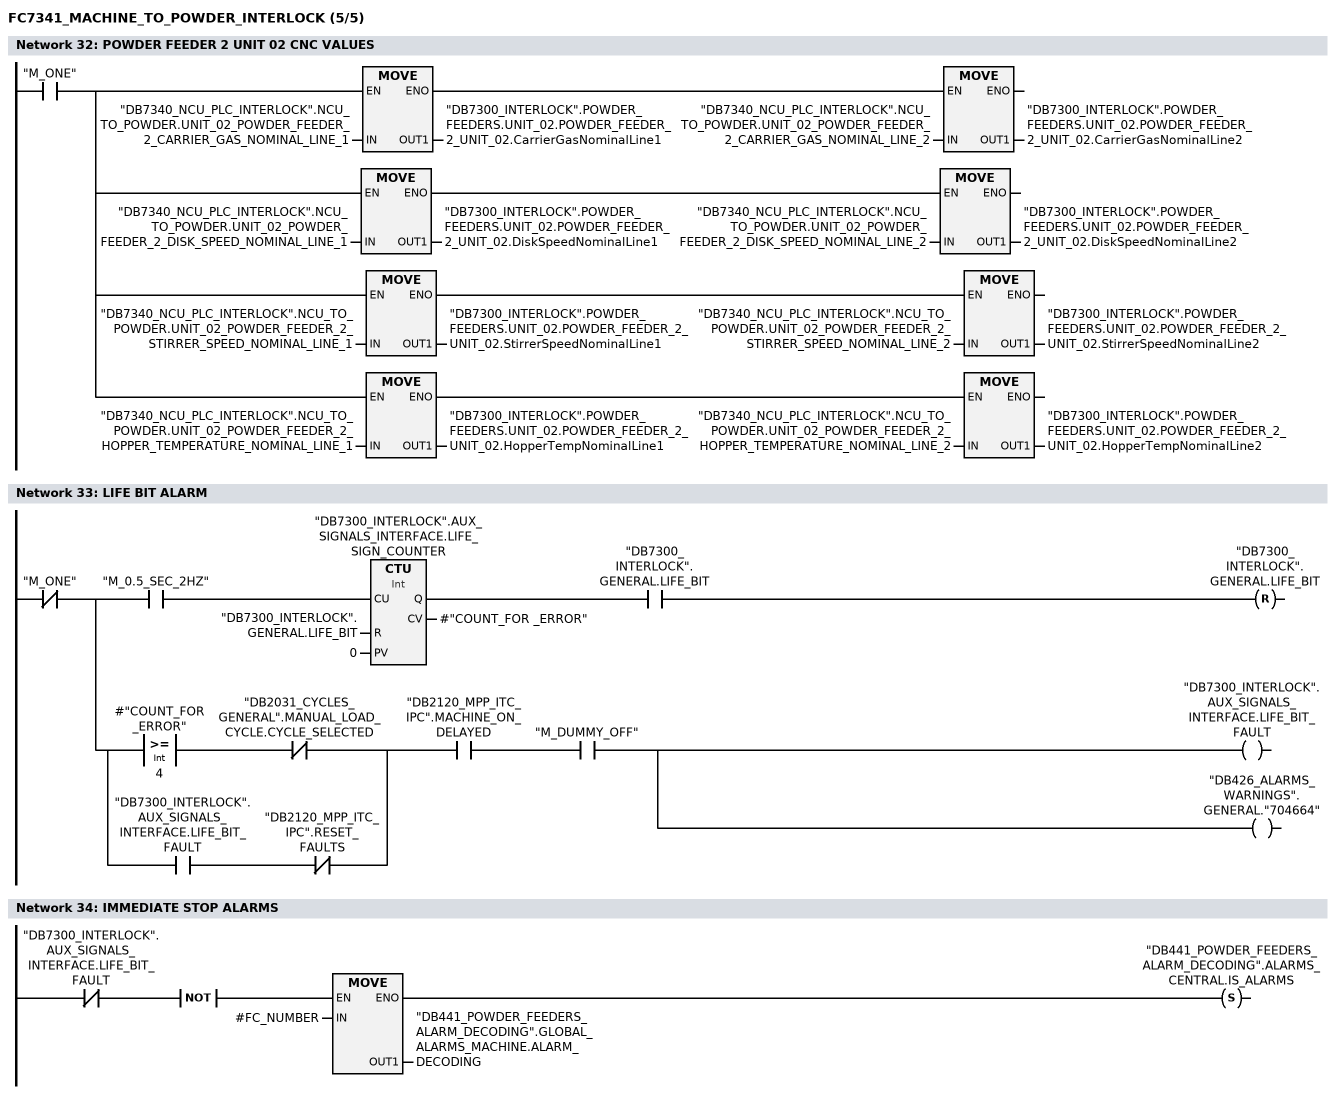
   RUNG wire#powerrail
      Contact( "M_ONE" )
      wire#w1
      Move(in := "DB7340_NCU_PLC_INTERLOCK".NCU_TO_POWDER.UNIT_02_POWDER_FEEDER_2_CARRIER_GAS_NOMINAL_LINE_1, out1 => "DB7300_INTERLOCK".POWDER_FEEDERS.UNIT_02.POWDER_FEEDER_2_UNIT_02.CarrierGasNominalLine1)
      Move(in := "DB7340_NCU_PLC_INTERLOCK".NCU_TO_POWDER.UNIT_02_POWDER_FEEDER_2_CARRIER_GAS_NOMINAL_LINE_2, out1 => "DB7300_INTERLOCK".POWDER_FEEDERS.UNIT_02.POWDER_FEEDER_2_UNIT_02.CarrierGasNominalLine2)
   END_RUNG
   RUNG wire#w1
      Move(in := "DB7340_NCU_PLC_INTERLOCK".NCU_TO_POWDER.UNIT_02_POWDER_FEEDER_2_DISK_SPEED_NOMINAL_LINE_1, out1 => "DB7300_INTERLOCK".POWDER_FEEDERS.UNIT_02.POWDER_FEEDER_2_UNIT_02.DiskSpeedNominalLine1)
      Move(in := "DB7340_NCU_PLC_INTERLOCK".NCU_TO_POWDER.UNIT_02_POWDER_FEEDER_2_DISK_SPEED_NOMINAL_LINE_2, out1 => "DB7300_INTERLOCK".POWDER_FEEDERS.UNIT_02.POWDER_FEEDER_2_UNIT_02.DiskSpeedNominalLine2)
   END_RUNG
   RUNG wire#w1
      Move(in := "DB7340_NCU_PLC_INTERLOCK".NCU_TO_POWDER.UNIT_02_POWDER_FEEDER_2_STIRRER_SPEED_NOMINAL_LINE_1, out1 => "DB7300_INTERLOCK".POWDER_FEEDERS.UNIT_02.POWDER_FEEDER_2_UNIT_02.StirrerSpeedNominalLine1)
      Move(in := "DB7340_NCU_PLC_INTERLOCK".NCU_TO_POWDER.UNIT_02_POWDER_FEEDER_2_STIRRER_SPEED_NOMINAL_LINE_2, out1 => "DB7300_INTERLOCK".POWDER_FEEDERS.UNIT_02.POWDER_FEEDER_2_UNIT_02.StirrerSpeedNominalLine2)
   END_RUNG
   RUNG wire#w1
      Move(in := "DB7340_NCU_PLC_INTERLOCK".NCU_TO_POWDER.UNIT_02_POWDER_FEEDER_2_HOPPER_TEMPERATURE_NOMINAL_LINE_1, out1 => "DB7300_INTERLOCK".POWDER_FEEDERS.UNIT_02.POWDER_FEEDER_2_UNIT_02.HopperTempNominalLine1)
      Move(in := "DB7340_NCU_PLC_INTERLOCK".NCU_TO_POWDER.UNIT_02_POWDER_FEEDER_2_HOPPER_TEMPERATURE_NOMINAL_LINE_2, out1 => "DB7300_INTERLOCK".POWDER_FEEDERS.UNIT_02.POWDER_FEEDER_2_UNIT_02.HopperTempNominalLine2)
   END_RUNG
   // the same network as SCL:
   IF "M_ONE" THEN
       "DB7300_INTERLOCK".POWDER_FEEDERS.UNIT_02.POWDER_FEEDER_2_UNIT_02.CarrierGasNominalLine1 := "DB7340_NCU_PLC_INTERLOCK".NCU_TO_POWDER.UNIT_02_POWDER_FEEDER_2_CARRIER_GAS_NOMINAL_LINE_1;
       "DB7300_INTERLOCK".POWDER_FEEDERS.UNIT_02.POWDER_FEEDER_2_UNIT_02.CarrierGasNominalLine2 := "DB7340_NCU_PLC_INTERLOCK".NCU_TO_POWDER.UNIT_02_POWDER_FEEDER_2_CARRIER_GAS_NOMINAL_LINE_2;
       "DB7300_INTERLOCK".POWDER_FEEDERS.UNIT_02.POWDER_FEEDER_2_UNIT_02.DiskSpeedNominalLine1 := "DB7340_NCU_PLC_INTERLOCK".NCU_TO_POWDER.UNIT_02_POWDER_FEEDER_2_DISK_SPEED_NOMINAL_LINE_1;
       "DB7300_INTERLOCK".POWDER_FEEDERS.UNIT_02.POWDER_FEEDER_2_UNIT_02.DiskSpeedNominalLine2 := "DB7340_NCU_PLC_INTERLOCK".NCU_TO_POWDER.UNIT_02_POWDER_FEEDER_2_DISK_SPEED_NOMINAL_LINE_2;
       "DB7300_INTERLOCK".POWDER_FEEDERS.UNIT_02.POWDER_FEEDER_2_UNIT_02.StirrerSpeedNominalLine1 := "DB7340_NCU_PLC_INTERLOCK".NCU_TO_POWDER.UNIT_02_POWDER_FEEDER_2_STIRRER_SPEED_NOMINAL_LINE_1;
       "DB7300_INTERLOCK".POWDER_FEEDERS.UNIT_02.POWDER_FEEDER_2_UNIT_02.StirrerSpeedNominalLine2 := "DB7340_NCU_PLC_INTERLOCK".NCU_TO_POWDER.UNIT_02_POWDER_FEEDER_2_STIRRER_SPEED_NOMINAL_LINE_2;
       "DB7300_INTERLOCK".POWDER_FEEDERS.UNIT_02.POWDER_FEEDER_2_UNIT_02.HopperTempNominalLine1 := "DB7340_NCU_PLC_INTERLOCK".NCU_TO_POWDER.UNIT_02_POWDER_FEEDER_2_HOPPER_TEMPERATURE_NOMINAL_LINE_1;
       "DB7300_INTERLOCK".POWDER_FEEDERS.UNIT_02.POWDER_FEEDER_2_UNIT_02.HopperTempNominalLine2 := "DB7340_NCU_PLC_INTERLOCK".NCU_TO_POWDER.UNIT_02_POWDER_FEEDER_2_HOPPER_TEMPERATURE_NOMINAL_LINE_2;
   END_IF;
END_REGION

REGION Network 33: LIFE BIT ALARM
   RUNG wire#powerrail
      I_Contact( "M_ONE" )
      wire#w1
      Contact( "M_0.5_SEC_2HZ" )
      { S7_Templates := "value_type := Int" } "DB7300_INTERLOCK".AUX_SIGNALS_INTERFACE.LIFE_SIGN_COUNTER.CTU(r := "DB7300_INTERLOCK".GENERAL.LIFE_BIT, pv := 0, cv => #"COUNT_FOR _ERROR")
      Contact( "DB7300_INTERLOCK".GENERAL.LIFE_BIT )
      R_Coil( "DB7300_INTERLOCK".GENERAL.LIFE_BIT )
   END_RUNG
   RUNG wire#w1
      { S7_Templates := "SrcType := Int" } GE_Contact(in1 := #"COUNT_FOR _ERROR", in2 := 4)
      I_Contact( "DB2031_CYCLES_GENERAL".MANUAL_LOAD_CYCLE.CYCLE_SELECTED )
      wire#w2
      Contact( "DB2120_MPP_ITC_IPC".MACHINE_ON_DELAYED )
      Contact( "M_DUMMY_OFF" )
      wire#w3
      Coil( "DB7300_INTERLOCK".AUX_SIGNALS_INTERFACE.LIFE_BIT_FAULT )
   END_RUNG
   RUNG wire#w1
      Contact( "DB7300_INTERLOCK".AUX_SIGNALS_INTERFACE.LIFE_BIT_FAULT )
      I_Contact( "DB2120_MPP_ITC_IPC".RESET_FAULTS )
   END_RUNG wire#w2
   RUNG wire#w3
      Coil( "DB426_ALARMS_WARNINGS".GENERAL."704664" )
   END_RUNG
   // the same network as SCL:
   "DB7300_INTERLOCK".AUX_SIGNALS_INTERFACE.LIFE_SIGN_COUNTER.CTU(CU := NOT "M_ONE" AND "M_0.5_SEC_2HZ",
                           R := "DB7300_INTERLOCK".GENERAL.LIFE_BIT,
                           PV := 0,
                           CV => #"COUNT_FOR _ERROR");
   IF "DB7300_INTERLOCK".AUX_SIGNALS_INTERFACE.LIFE_SIGN_COUNTER.Q AND "DB7300_INTERLOCK".GENERAL.LIFE_BIT THEN
       "DB7300_INTERLOCK".GENERAL.LIFE_BIT := FALSE;
   END_IF;
   "DB7300_INTERLOCK".AUX_SIGNALS_INTERFACE.LIFE_BIT_FAULT := NOT "M_ONE" AND (((#"COUNT_FOR _ERROR" >= 4) AND NOT "DB2031_CYCLES_GENERAL".MANUAL_LOAD_CYCLE.CYCLE_SELECTED) OR ("DB7300_INTERLOCK".AUX_SIGNALS_INTERFACE.LIFE_BIT_FAULT AND NOT "DB2120_MPP_ITC_IPC".RESET_FAULTS)) AND "DB2120_MPP_ITC_IPC".MACHINE_ON_DELAYED AND "M_DUMMY_OFF";
   "DB426_ALARMS_WARNINGS".GENERAL."704664" := "DB7300_INTERLOCK".AUX_SIGNALS_INTERFACE.LIFE_BIT_FAULT;
END_REGION

REGION Network 34: IMMEDIATE STOP ALARMS
   RUNG wire#powerrail
      I_Contact( "DB7300_INTERLOCK".AUX_SIGNALS_INTERFACE.LIFE_BIT_FAULT )
      Not()
      { S7_GenerateENO := "TRUE" } Move(in := #FC_NUMBER, out1 => "DB441_POWDER_FEEDERS_ALARM_DECODING".GLOBAL_ALARMS_MACHINE.ALARM_DECODING)
      S_Coil( "DB441_POWDER_FEEDERS_ALARM_DECODING".ALARMS_CENTRAL.IS_ALARMS )
   END_RUNG
   // the same network as SCL:
   // ENO of a box is taken as its EN; it also drops when the box reports an error
   IF NOT (NOT "DB7300_INTERLOCK".AUX_SIGNALS_INTERFACE.LIFE_BIT_FAULT) THEN
       "DB441_POWDER_FEEDERS_ALARM_DECODING".GLOBAL_ALARMS_MACHINE.ALARM_DECODING := #FC_NUMBER;
       "DB441_POWDER_FEEDERS_ALARM_DECODING".ALARMS_CENTRAL.IS_ALARMS := TRUE;
   END_IF;
END_REGION
END_FUNCTION
